// TwinCAT 3 PLC project PLC1
// ProgramVersion: 3.1.4024.0
// libraries:
//   Tc2_Standard, * (Beckhoff Automation GmbH)
//   Tc2_System, * (Beckhoff Automation GmbH)
//   Tc2_Utilities, * (Beckhoff Automation GmbH)
//   Tc3_IotBase, * (Beckhoff Automation GmbH)
//   Tc3_Module, * (Beckhoff Automation GmbH)
//   Util, * (System)
// project tree:
//   CSL/Enums/ E_Step.TcTLEO
//   CSL/FB/IO/ FB_UpdateInputs.TcPOU, FB_UpdateOutputs.TcPOU, FB_UpdatesParams.TcPOU
//   CSL/FB/Main/ FB_CSL_MAIN.TcPOU, FB_Oscillator.TcPOU, FB_Restore.TcPOU
//   CSL/FB/Piston/ FB_MSF_Pistons.TcPOU
//   CSL/FB/Sensor/ FB_Filter.TcPOU (not stored), FB_Measuring.TcPOU, FB_MSF_Sensor.TcPOU, FB_Processing.TcPOU
//   CSL/FC/ FC_Conversion.TcPOU, FC_thresholdsCalculation.TcPOU
//   CSL/Structs/ ST_CSL_RawOut.TcDUT (not stored), ST_CSL_In.TcDUT (not stored), ST_CSL_Out.TcDUT (not stored), ST_CSL_Params.TcDUT, ST_CSL_RawIn.TcDUT, ST_HMI_In.TcDUT, ST_HMI_Out.TcDUT, ST_HMI_Params.TcDUT
//   GVLs/ GVL_IOT.TcGVL, GVL_PLC.TcGVL
//   / IoTTask.TcTTO, PlcTask.TcTTO
//   IOT/Enums/ E_IOT_DataType.TcDUT, E_IOT_Step.TcDUT, E_IOT_UpdateSpeed.TcDUT
//   IOT/ FB_IOT.TcPOU, GVL_IOT_Constants.TcGVL
//   IOT/Functions/ F_IOT_GetPayload.TcPOU, F_IOT_IsValueEqual.TcPOU
//   IOT/Structs/ ST_IOT_Data.TcDUT, ST_IOT_OnChangePublishData.TcDUT, ST_IOT_Params.TcDUT, ST_IOT_PeriodicPublishData.TcDUT
//   IOT/Unions/ U_IOT_DataValue.TcDUT
//   POUs/ IOT_MAIN.TcPOU, MAIN.TcPOU
// real-time tasks:
//   TASK PlcTask: cycle T#10ms, priority 20, ADS port 350
//   TASK IoTTask: cycle T#10ms, priority 21, ADS port 351
// motion (NC):
//   TASK NC-Task 1 SAF: cycle T#2ms, priority 4, ADS port 501
//   TASK NC-Task 1 SVB: cycle T#10ms, priority 8, ADS port 511
//   AXIS Asse 1 (id 1)
//     OtherSettings: AllowMotionCmdToSlave=true
//     encoder EncType=4
//       EncPara: MaxCount=#x0000ffff
//         Inc: RefSoftSyncMask=#x0000ffff
//     drive DrvType=24
//       Analog: TorqueSetpointScale=10, ScaleFactorActTorque=0.1
//       TimeComp: TaskDelayCycles=1
//     controller CtrType=1
//       CtrPara: PriorControlFactor=1
//         Observer: BandWidth=20
//   AXIS Asse 2 (id 2)
//     OtherSettings: AllowMotionCmdToSlave=true
//     encoder EncType=4
//       EncPara: MaxCount=#x0000ffff
//         Inc: RefSoftSyncMask=#x0000ffff
//     drive DrvType=24
//       Analog: TorqueSetpointScale=10, ScaleFactorActTorque=0.1
//       TimeComp: TaskDelayCycles=1
//     controller CtrType=1
//       CtrPara: PriorControlFactor=1
//         Observer: BandWidth=20
//   AXIS Asse 3 (id 3)
//     OtherSettings: AllowMotionCmdToSlave=true
//     encoder EncType=4
//       EncPara: MaxCount=#x0000ffff
//         Inc: RefSoftSyncMask=#x0000ffff
//     drive DrvType=24
//       Analog: TorqueSetpointScale=10, ScaleFactorActTorque=0.1
//       TimeComp: TaskDelayCycles=1
//     controller CtrType=1
//       CtrPara: PriorControlFactor=1
//         Observer: BandWidth=20
// I/O:
//   DEVICE Dispositivo 1 (EtherCAT), AmsNetId 5.85.197.242.2.1
//     Terminale 1 (EK1200) [EK1200-5000 EtherCAT Power supply (2A E-Bus)]
//       Terminale 2 (EL1809) [EL1809 16Ch. Dig. Input 24V, 3ms]
//       Terminale 3 (EL2809) [EL2809 16Ch. Dig. Output 24V, 0.5A]
//       Terminale 4 (EL3201) [EL3201 1Ch. Ana. Input PT100 (RTD)]
//       Terminale 5 (EL3311) [EL3311 1Ch. Ana. Input Thermocouple (TC)]
//       Terminale 6 (EL3004) [EL3004 4Ch. Ana. Input +/-10V]
//       Terminale 7 (EL1918) [EL1918, 8Ch. Safety Input 24V, TwinSAFE]
//         modules: Module 1 (FSOE), Module 2 (FSLOGIC)
//       Terminale 8 (EL2904) [EL2904, 4 Ch. Safety Output 24V, 0.5A, TwinSAFE]
//         modules: Module 1 (FSOES), Module 2 (DO)
//       Terminale 9 (EL9011) [EL9011 End Terminal]
//   DEVICE Dispositivo 4 (EtherCAT), AmsNetId 5.85.197.242.5.1
//     Terminale 10 (EK1100) [EK1100 EtherCAT Coupler (2A E-Bus)]
//       Terminale 11 (EL1809) [EL1809 16Ch. Dig. Input 24V, 3ms]
//       Terminale 12 (EL2809) [EL2809 16Ch. Dig. Output 24V, 0.5A]
//       Terminale 13 (EL1809) [EL1809 16Ch. Dig. Input 24V, 3ms]
//       Terminale 14 (EL2809-0015) [EL2809-0015 16Ch. Dig. Output 24V DC, 0.35A, not short-circuit proof]
//       Terminale 15 (EL3202) [EL3202 2Ch. Ana. Input PT100 (RTD)]
//       Terminale 16 (EL3312) [EL3312 2Ch. Ana. Input Thermocouple (TC)]
//       Terminale 17 (EL3632) [EL3632 2Ch. IEPE Sensor]
//       Terminale 18 (EL7031) [EL7031 1Ch. Stepper motor output stage (24V, 1.5A)]
//       Terminale 10 (EL9011) [EL9011 End Terminal]
// variable links:
//   NC-Task 1 SAF/Axes/Asse 3 <-> Device 4 (EtherCAT)/Term 10 (EK1100)/Term 18 (EL7031)
//     Drive/Inputs/In/nState1 @bit 3 <-> STM Status/Status/Error
//     Drive/Inputs/In/nState1 @bit 5 <-> STM Status/Status/Moving negative
//     Drive/Inputs/In/nState1 @bit 4 <-> STM Status/Status/Moving positive
//     Drive/Inputs/In/nState1 @bit 1 <-> STM Status/Status/Ready
//     Drive/Inputs/In/nState1 <-> STM Status/Status/Ready to enable
//     Drive/Inputs/In/nState1 @bit 6 <-> STM Status/Status/Torque reduced
//     Drive/Inputs/In/nState1 @bit 2 <-> STM Status/Status/Warning
//     Drive/Inputs/In/nState2 @bit 3 <-> STM Status/Status/Digital input 1
//     Drive/Inputs/In/nState2 @bit 4 <-> STM Status/Status/Digital input 2
//     Drive/Inputs/In/nState2 @bit 5 <-> STM Status/Status/Sync error
//     Drive/Inputs/In/nState2 @bit 7 <-> STM Status/Status/TxPDO Toggle
//     Drive/Inputs/In/nState4 @bit 1 <-> WcState/InputToggle
//     Drive/Inputs/In/nState4 <-> WcState/WcState
//     Drive/Outputs/Out/nCtrl1 <-> STM Control/Control/Enable
//     Drive/Outputs/Out/nCtrl1 @bit 2 <-> STM Control/Control/Reduce torque
//     Drive/Outputs/Out/nCtrl1 @bit 1 <-> STM Control/Control/Reset
//     Drive/Outputs/Out/nDataOut2[0] <-> STM Velocity/Velocity
//     Enc/Inputs/In/nDataIn1[0] <-> ENC Status compact/Counter value
//     Enc/Inputs/In/nDataIn2[0] <-> ENC Status compact/Latch value
//     Enc/Inputs/In/nState1 @bit 4 <-> ENC Status compact/Status/Counter overflow
//     Enc/Inputs/In/nState1 @bit 3 <-> ENC Status compact/Status/Counter underflow
//     Enc/Inputs/In/nState1 @bit 1 <-> ENC Status compact/Status/Latch extern valid
//     Enc/Inputs/In/nState1 @bit 2 <-> ENC Status compact/Status/Set counter done
//     Enc/Inputs/In/nState2 @bit 4 <-> ENC Status compact/Status/Status of extern latch
//     Enc/Inputs/In/nState2 @bit 5 <-> ENC Status compact/Status/Sync error
//     Enc/Inputs/In/nState2 @bit 7 <-> ENC Status compact/Status/TxPDO Toggle
//     Enc/Inputs/In/nState4 @bit 1 <-> WcState/InputToggle
//     Enc/Inputs/In/nState4 <-> WcState/WcState
//     Enc/Outputs/Out/nCtrl1 @bit 3 <-> ENC Control compact/Control/Enable latch extern on negative edge
//     Enc/Outputs/Out/nCtrl1 @bit 1 <-> ENC Control compact/Control/Enable latch extern on positive edge
//     Enc/Outputs/Out/nCtrl1 @bit 2 <-> ENC Control compact/Control/Set counter
//     Enc/Outputs/Out/nDataOut1[0] <-> ENC Control compact/Set counter value
//   PLC1/PLC1 Instance <-> Device 1 (EtherCAT)/Term 1 (EK1200)/Term 2 (EL1809)
//     PlcTask Inputs/MAIN.stRawIn.bAck <-> Channel 10/Input
//     PlcTask Inputs/MAIN.stRawIn.bEmerg <-> Channel 11/Input
//     PlcTask Inputs/MAIN.stRawIn.bMotorImpulse <-> Channel 1/Input
//     PlcTask Inputs/MAIN.stRawIn.bPieceSensorInput <-> Channel 2/Input
//     PlcTask Inputs/MAIN.stRawIn.bPieceSensorOutput <-> Channel 3/Input
//     PlcTask Inputs/MAIN.stRawIn.bSlot1 <-> Channel 5/Input
//     PlcTask Inputs/MAIN.stRawIn.bSlot2 <-> Channel 6/Input
//     PlcTask Inputs/MAIN.stRawIn.bSlot3 <-> Channel 7/Input
//     PlcTask Inputs/MAIN.stRawIn.bStart <-> Channel 8/Input
//     PlcTask Inputs/MAIN.stRawIn.bStop <-> Channel 9/Input
//   PLC1/PLC1 Instance <-> Device 1 (EtherCAT)/Term 1 (EK1200)/Term 3 (EL2809)
//     PlcTask Outputs/MAIN.stRawOut.bCompressor <-> Channel 2/Output
//     PlcTask Outputs/MAIN.stRawOut.bLAck <-> Channel 8/Output
//     PlcTask Outputs/MAIN.stRawOut.bLStart <-> Channel 6/Output
//     PlcTask Outputs/MAIN.stRawOut.bLStop <-> Channel 7/Output
//     PlcTask Outputs/MAIN.stRawOut.bMotor <-> Channel 1/Output
//     PlcTask Outputs/MAIN.stRawOut.bValveSlot1 <-> Channel 3/Output
//     PlcTask Outputs/MAIN.stRawOut.bValveSlot2 <-> Channel 4/Output
//     PlcTask Outputs/MAIN.stRawOut.bValveSlot3 <-> Channel 5/Output
//   PLC1/PLC1 Instance <-> Device 1 (EtherCAT)/Term 1 (EK1200)/Term 6 (EL3004)
//     PlcTask Inputs/MAIN.stRawIn.nColorSensor <-> AI Standard Channel 1/Value

CONFIGURATION PLC1
    RESOURCE PLC ON TwinCAT3
        TASK IoTTask(INTERVAL := T#10ms, PRIORITY := 21);
        TASK PlcTask(INTERVAL := T#10ms, PRIORITY := 20);
        PROGRAM IOT_MAIN WITH IoTTask : IOT_MAIN;
        PROGRAM MAIN WITH PlcTask : MAIN;
    END_RESOURCE
END_CONFIGURATION

// ---- CSL/Enums/E_Step.TcTLEO
{attribute 'qualified_only'}
{attribute 'strict'}
{attribute 'to_string'}
TYPE E_Step :
(
	(* special steps *)
	NoStep := -32767,  // No step   
	Unknown := -32000, // unknown step
	
	(* Not Enabled or Errors*)    
	NeOrError := -990, // Not Enabled or Errors
	
	(*MSF Steps*)
	//main steps
	MainStop 		:= 	10, 		// stop
	MainSensor		:=	20,		// sensor area
	MainPiston		:=	30,		// piston area
	MainPause		:=	40,		// pause
	MainEmergency	:=	50,		// emergency
	MainAcknowledge	:=	60,		// acknowledge
	//sub-steps
	Stop			:=  90,
	Start			:= 	100,
	Measuring		:= 	110,
	Processing		:= 	120,
	conveyor		:=  130,	// a new piece was placed on the conveyor belt
	waiting			:= 	140,	// attesa
	piston			:=	150		// pistone

);
END_TYPE
//  NoStep = '-32767'
//  Unknown = '-32000'
//  NeOrError = '-990'

// ---- CSL/Structs/ST_CSL_Params.TcDUT
TYPE ST_CSL_Params :
STRUCT
	StepSlot1			:	INT		:= 	3;  // conveyor steps to reach Slot 1
	StepSlot2			:	INT		:= 	8;  // conveyor steps to reach Slot 2
	StepSlot3			:	INT		:= 	13; // conveyor steps to reach Slot 3
	StepNoSlot			:	INT		:=	20; // unknown colour -> discard piece
		
	pistonReentryDelay	:	TIME	:= T#500MS; // piston re-entry time
	stopLongPressTime	:	TIME	:= T#500MS;	// time required for the pause transition to be activated
	slotRemoveTime		:	TIME	:= T#500MS; // time required after piece removal from its slot
	
	(*Colors Voltage*)
	RedVoltage			:	REAL;	//	:=	5.5;
	BlueVoltage			:	REAL;	//	:=	7.1;
	WhiteVoltage		:	REAL;	//	:=	2.9;
	
	//threshold
	Threshold			:	REAL;	//	:=	0.5;
	
	//min values
	RedVoltageMin		:	REAL;
	BlueVoltageMin		:	REAL;
	WhiteVoltageMin		:	REAL;
	
	//max values
	RedVoltageMax		:	REAL;
	BlueVoltageMax		:	REAL;
	WhiteVoltageMax		:	REAL;
	
	(*Colors Slot*)
	WhiteSlot			:	INT;	//	:=	1;
	BlueSlot			:	INT;	//	:=	2;
	RedSlot				:	INT;	//	:=	3;

END_STRUCT
END_TYPE

// ---- CSL/Structs/ST_CSL_RawIn.TcDUT
TYPE ST_CSL_RawIn :
STRUCT
	(*Digital Inputs*)
	bMotorImpulse 		AT %I*	:	BOOL;	//I1  (NC)
	bPieceSensorInput 	AT %I*	:	BOOL;	//I2  (NC)
	bPieceSensorOutput 	AT %I*	:	BOOL;	//I3  (NO)
	bSlot1 				AT %I*	:	BOOL;	//I5  (NC)
	bSlot2 				AT %I*	:	BOOL;	//I6  (NC)
	bSlot3				AT %I*	:	BOOL;	//I7  (NC)
	
	bStart 				AT %I*	:	BOOL;	//I9  (NO)
	bStop				AT %I*	:	BOOL;	//I10 (NC)
	bAck 				AT %I*	:	BOOL;	//I11 (NO)
	bEmerg 				AT %I*	:	BOOL;	//I12 (NC)
	bMainEmerg			AT %I*	:	BOOL;	//I13 (NC)
	
	(*Analog Input*)
	nColorSensor		AT %I*	:	INT;	//I4
END_STRUCT
END_TYPE

// ---- CSL/Structs/ST_HMI_In.TcDUT
TYPE ST_HMI_In :
STRUCT
	bStart 		:	BOOL;
	bStop 		:	BOOL;
	bAck		:	BOOL;
END_STRUCT
END_TYPE

// ---- CSL/Structs/ST_HMI_Out.TcDUT
TYPE ST_HMI_Out :
STRUCT
	bGreen	:BOOL;
	bRed	:BOOL;
	bOrange	:BOOL;
END_STRUCT
END_TYPE

// ---- CSL/Structs/ST_HMI_Params.TcDUT
TYPE ST_HMI_Params :
STRUCT
	(*Params*)
	//slot
	WhiteSlot		:	INT	:= 1;
	BlueSlot		:	INT	:= 2;
	RedSlot			:	INT := 3;
	
	//voltage levels
	RedVoltage		:	REAL	:= 5.5;
	BlueVoltage		:	REAL	:= 7.1;
	WhiteVoltage	:	REAL	:= 2.9;
	
	//threshold
	Threshold		:	REAL	:=	0.5;
END_STRUCT
END_TYPE

// ---- IOT/Enums/E_IOT_DataType.TcDUT
(* -----------------------------------------------------------------------------
| This sample has been supplied by Beckhoff As-Is and is intended only as an   |
| example implementation. Functionality is not guaranteed.                     |
----------------------------------------------------------------------------- *)

// questa enumerazione descrive serve per identificare il tipo di dato contenuto
// all'interno dell'unione U_IOT_DataValue in modo da poterlo interpretare 
// correttamente

{attribute 'qualified_only'}
{attribute 'strict'}
TYPE E_IOT_DataType :
(
	Boolean := 0,
	I32 := 1,
	F64 := 2,
	S50 := 51
);
END_TYPE

// ---- IOT/Enums/E_IOT_Step.TcDUT
(* -----------------------------------------------------------------------------
| This sample has been supplied by Beckhoff As-Is and is intended only as an   |
| example implementation. Functionality is not guaranteed.                     |
----------------------------------------------------------------------------- *)

// passi della macchina a stati che gestisce la comunicazione IOT

{attribute 'qualified_only'}
{attribute 'strict'}
TYPE E_IOT_Step :
(
	(* special steps *)
	NoStep := -32767,		// nessuno step
	Unknown := -32000,		// step sconosciuto
	
	(* Error steps *)
	NeOrError := -990,		// non abilitata o in errore
	Reset := -980,			// azzeramento errori

	(* Stop *)
	Stop := 0,				// stop
	
	(* Cycle *)
	Configure := 100,		// configurazione 
	Connect := 200,			// connessione
	Subscribe := 210,		// sottoscrivi i topic che interessano
	Online := 220,			// in linea
	Unsubscribe := 300,		// rimuovi sottoscrizioni
	Disconnect := 310		// disconnessione
);
END_TYPE

// ---- IOT/Enums/E_IOT_UpdateSpeed.TcDUT
(* -----------------------------------------------------------------------------
| This sample has been supplied by Beckhoff As-Is and is intended only as an   |
| example implementation. Functionality is not guaranteed.                     |
----------------------------------------------------------------------------- *)

// questa enumerazione serve ad identificare il periodo di aggiornamento dei
// dati che vengono pubblicati su MQTT

{attribute 'qualified_only'}
{attribute 'strict'}
TYPE E_IOT_UpdateSpeed :
(
	Slow := 0,			// 1s	
	Fast := 1			// 100ms
);
END_TYPE

// ---- IOT/Structs/ST_IOT_Data.TcDUT
(* -----------------------------------------------------------------------------
| This sample has been supplied by Beckhoff As-Is and is intended only as an   |
| example implementation. Functionality is not guaranteed.                     |
----------------------------------------------------------------------------- *)

// Questa struttura definisce il dato da pubblicare sul broker
// Ad ogni dato viene associato un subtopic specifico

TYPE ST_IOT_Data :
STRUCT
	sSubtopic : STRING;				// subtopic dove il valore verra scritto
	eType : E_IOT_DataType;			// tipologia del dato (DINT, LREAL, BOOL)
	uValue : U_IOT_DataValue;		// unione in cui viene letto/scritto il valore	
END_STRUCT
END_TYPE

// ---- IOT/Structs/ST_IOT_OnChangePublishData.TcDUT
(* -----------------------------------------------------------------------------
| This sample has been supplied by Beckhoff As-Is and is intended only as an   |
| example implementation. Functionality is not guaranteed.                     |
----------------------------------------------------------------------------- *)

// Questa struttura definisce un dato da pubblicare al cambiamento del suo
// valore. Oltre al dato è presente nellea struttura l'elemento che su cui
// salvare il valore precedente in modo da poter fare dei confronti

TYPE ST_IOT_OnChangePublishData :
STRUCT
	uOldValue : U_IOT_DataValue;
	stData : ST_IOT_Data;		
END_STRUCT
END_TYPE

// ---- IOT/Structs/ST_IOT_Params.TcDUT
(* -----------------------------------------------------------------------------
| This sample has been supplied by Beckhoff As-Is and is intended only as an   |
| example implementation. Functionality is not guaranteed.                     |
----------------------------------------------------------------------------- *)

// Questa struttura cointiene i parametri necessari al funzionamento della
// FB_IOT. 

TYPE ST_IOT_Params :
STRUCT
	// i parametri per instaurare la connessione con il broker 
	//sHostName : STRING := 'test.mosquitto.org';
	sMQTTHostName : STRING := 'item2122a.cloud.shiftr.io';
	nHostPort : UINT := 1883; 
	// Si possono usare anche user e password. 
    // vd: https://infosys.beckhoff.com/content/1033/tf6701_tc3_iot_communication_mqtt/3391835403.html?id=6531035858226877065
	sUserName : STRING := 'item2122a';
	sUserPassword : STRING := 'K2Xpe5XV3yvL7zcu';
	
	// certificati necessari per l'autenticazione. 
	stMqttTls : ST_IotMqttTls := ();
		
	// topic generale all'interno del quale ci saranno i subtopic nei quali
	// verranno pubblicati i dati
	// il pragma {attribute 'TcEncoding':='UTF-8'} va sempre usato per le 
	// stringhe quando si opera con MQTT
	{attribute 'TcEncoding':='UTF-8'}
	sTopicPrefix : STRING := 'ColorSorter';
	
	// subtopic da sottoscrivere per leggere i comandi  
	{attribute 'TcEncoding':='UTF-8'}
	sCmdSubscribedTopic : STRING := '/cmd';
	
	// numero massimo di messaggi da leggere per ciclo dai topic sottoscritti 
	nDequeueMessagesPerCycle : UINT := 3;
END_STRUCT
END_TYPE

// ---- IOT/Structs/ST_IOT_PeriodicPublishData.TcDUT
(* -----------------------------------------------------------------------------
| This sample has been supplied by Beckhoff As-Is and is intended only as an   |
| example implementation. Functionality is not guaranteed.                     |
----------------------------------------------------------------------------- *)

// Questa struttura definisce un dato da pubblicare ciclicamente. Oltre al 
// dato è presente nellea struttura l'elemento che definisce l'intervallo 
// di pubblicazione

TYPE ST_IOT_PeriodicPublishData :
STRUCT
	eUpdateSpeed : E_IOT_UpdateSpeed;
	stData : ST_IOT_Data;	
END_STRUCT
END_TYPE

// ---- IOT/Unions/U_IOT_DataValue.TcDUT
(* -----------------------------------------------------------------------------
| This sample has been supplied by Beckhoff As-Is and is intended only as an   |
| example implementation. Functionality is not guaranteed.                     |
----------------------------------------------------------------------------- *)

// Questa unione contiene il valore del dato. L'utilizzo dell'unione permette
// di avere una struttura dato (ST_IOT_Data) generica evitando di preoccuparsi 
// di quale sia il tipo di dato contenuto se non quando si va effettivamente 
// a leggerlo o scriverlo.
// La quantità di memoria occupata da una union corrisponde alla quantita di 
// memoria necessaria a contenere l'elemento della union che da dimensione
// maggiore.
// In sostanza i vari elementi di una union condividono la stessa area di
// memoria e usarne uno piuttosto di un altro non modifica il contenuto della
// memoria stessa quanto la sua rappresentazione.

TYPE U_IOT_DataValue :
UNION
	b : BOOL;
	n : DINT;
	f : LREAL;
	sv : STRING(50);
END_UNION
END_TYPE

// ---- GVLs/GVL_IOT.TcGVL
(* -----------------------------------------------------------------------------
| This sample has been supplied by Beckhoff As-Is and is intended only as an   |
| example implementation. Functionality is not guaranteed.                     |
----------------------------------------------------------------------------- *)

{attribute 'qualified_only'}
VAR_GLOBAL PERSISTENT
	stIotParams : ST_IOT_Params;		// Parametri per la comunicazione MQTT
//	stFlmCmd : ST_FLM_Cmd;				// comandi di FLM
END_VAR

// ---- GVLs/GVL_PLC.TcGVL
{attribute 'qualified_only'}
VAR_GLOBAL
	strEStep	:	STRING;
	strEsubStepSensor	:	STRING;
	strEsubStepPiston	:	STRING;
	
	estep 	: E_Step;
	eSubStepSensor: E_Step;
	eSubStepPistons: E_Step;
	
	nColorSensor	:	REAL;
	
	nTotalRevs		:	REAL;
	
	nCycles			:	INT;
END_VAR

// ---- IOT/GVL_IOT_Constants.TcGVL
(* -----------------------------------------------------------------------------
| This sample has been supplied by Beckhoff As-Is and is intended only as an   |
| example implementation. Functionality is not guaranteed.                     |
----------------------------------------------------------------------------- *)


{attribute 'qualified_only'}
VAR_GLOBAL CONSTANT
	cIOTMAXDATA : UDINT := 32;
END_VAR

// ---- POUs/IOT_MAIN.TcPOU
(* -----------------------------------------------------------------------------
| This sample has been supplied by Beckhoff As-Is and is intended only as an   |
| example implementation. Functionality is not guaranteed.                     |
----------------------------------------------------------------------------- *)

PROGRAM IOT_MAIN
VAR
	bInitialized : BOOL;
	bConnect : BOOL;		// richiesta TRUE -> connetti FALSE -> disconnetti
	
	// array per i dati da pubblicare e loro dimensione 
	aPeriodicPublish : ARRAY[0..GVL_IOT_Constants.cIOTMAXDATA - 1] OF ST_IOT_PeriodicPublishData;
	aOnChangePublish : ARRAY[0..GVL_IOT_Constants.cIOTMAXDATA - 1] OF ST_IOT_OnChangePublishData;		
	nPeriodicPublishSize : UDINT;	
	nOnChangePublishSize : UDINT;	
	
	fbIot : FB_IOT;
	nInitCycles : UDINT;
END_VAR

(* -----------------------------------------------------------------------------
| This sample has been supplied by Beckhoff As-Is and is intended only as an   |
| example implementation. Functionality is not guaranteed.                     |
----------------------------------------------------------------------------- *)

IF NOT bInitialized THEN
	IF nInitCycles = 0 THEN	
		ACT_InitPeriodic();	
		ACT_InitOnChange();
	END_IF;
	nInitCycles := nInitCycles + 1;
	bConnect := TRUE;
	bInitialized := (GVL_PLC.estep = E_Step.MainStop );
ELSE
	
	// Qui vengono letti ad ogni ciclo i valori da FLM che verranno pubblicati
	// nei topic corrispondenti
 
//	aOnChangePublish[0].stData.uValue.n := TO_DINT(GVL_PLC.stFlmStatus.eStep);
//	aOnChangePublish[1].stData.uValue.b := GVL_PLC.stFlmStatus.bFailure;
//	aOnChangePublish[2].stData.uValue.b := GVL_PLC.stFlmStatus.bWarning;

    aOnChangePublish[0].stData.uValue.f := TO_REAL(GVL_PLC.nColorSensor);
    aOnChangePublish[1].stData.uValue.sv := GVL_PLC.strEStep;
    aOnChangePublish[2].stData.uValue.sv := GVL_PLC.strEsubStepSensor;	
    aOnChangePublish[3].stData.uValue.sv := GVL_PLC.strEsubStepPiston;	
	aOnChangePublish[4].stData.uValue.f := GVL_PLC.nTotalRevs;	
	aOnChangePublish[5].stData.uValue.n := GVL_PLC.nCycles;
	
//	aPeriodicPublish[0].stData.uValue.b := GVL_PLC.stFlmOut.bCorkingVertical;

	
	fbIot(
		bEnable:= TRUE, 
		bConnect:= bConnect, 
		tAutoAckTime:= T#2M, 
		stParams:= GVL_IOT.stIotParams, 
		aPeriodicPublish := aPeriodicPublish,		
		aOnChangePublish := aOnChangePublish,
		nPeriodicPublishSize := nPeriodicPublishSize, 
		nOnChangePublishSize := nOnChangePublishSize
	);
	
	// I comandi letti nel subtopic corrispondente vengono qui scritti su
	// delle variabili globali in modo da poter essere letti dalla task PLC
	// e usati all'interno di FLM
//	GVL_IOT.stFlmCmd.bStart := fbIot.bFlmStartCmd;
//	GVL_IOT.stFlmCmd.bStop := fbIot.bFlmStopCmd;
//	GVL_IOT.stFlmCmd.bAck := fbIot.bFlmAckCmd;
END_IF

ACTION ACT_InitOnChange:
(* -----------------------------------------------------------------------------
| This sample has been supplied by Beckhoff As-Is and is intended only as an   |
| example implementation. Functionality is not guaranteed.                     |
----------------------------------------------------------------------------- *)

// inizializzazione degli elementi dell'array che contiene i dati da scambiare
// al cambiamento

aOnChangePublish[0].stData.sSubtopic := '/ncolorsensor';
aOnChangePublish[0].stData.eType := E_IOT_DataType.F64;

aOnChangePublish[1].stData.sSubtopic := '/estep';
aOnChangePublish[1].stData.eType := E_IOT_DataType.S50;

aOnChangePublish[2].stData.sSubtopic := '/esubstepsensor';
aOnChangePublish[2].stData.eType := E_IOT_DataType.S50;

aOnChangePublish[3].stData.sSubtopic := '/esubsteppistons';
aOnChangePublish[3].stData.eType := E_IOT_DataType.S50;

aOnChangePublish[4].stData.sSubtopic := '/nTotalRevs';
aOnChangePublish[4].stData.eType := E_IOT_DataType.F64;

aOnChangePublish[5].stData.sSubtopic := '/nCycles';
aOnChangePublish[5].stData.eType := E_IOT_DataType.I32;

//aOnChangePublish[2].stData.sSubtopic := '/Warning';
//aOnChangePublish[2].stData.eType := E_IOT_DataType.Boolean;

// dimensione effettiva dell'array
nOnChangePublishSize := 6;
END_ACTION

ACTION ACT_InitPeriodic:
(* -----------------------------------------------------------------------------
| This sample has been supplied by Beckhoff As-Is and is intended only as an   |
| example implementation. Functionality is not guaranteed.                     |
----------------------------------------------------------------------------- *)

// inizializzazione degli elementi dell'array che contiene i dati da scambiare
// ciclicamente.

aPeriodicPublish[0].eUpdateSpeed := E_IOT_UpdateSpeed.Fast;
aPeriodicPublish[0].stData.sSubtopic := '/TaskRunning';
aPeriodicPublish[0].stData.eType := E_IOT_DataType.Boolean;

(*
aPeriodicPublish[1].eUpdateSpeed := E_IOT_UpdateSpeed.Fast;
aPeriodicPublish[1].stData.sSubtopic := '/CorkingRotation';
aPeriodicPublish[1].stData.eType := E_IOT_DataType.Boolean;

aPeriodicPublish[2].eUpdateSpeed := E_IOT_UpdateSpeed.Slow;
aPeriodicPublish[2].stData.sSubtopic := '/WaterLevel';
aPeriodicPublish[2].stData.eType := E_IOT_DataType.F64;

aPeriodicPublish[3].eUpdateSpeed := E_IOT_UpdateSpeed.Slow;
aPeriodicPublish[3].stData.sSubtopic := '/MintLevel';
aPeriodicPublish[3].stData.eType := E_IOT_DataType.F64;
*)

// dimensione effettiva dell'array
nPeriodicPublishSize := 1;
END_ACTION

END_PROGRAM

// ---- IOT/FB_IOT.TcPOU
(* -----------------------------------------------------------------------------
| This sample has been supplied by Beckhoff As-Is and is intended only as an   |
| example implementation. Functionality is not guaranteed.                     |
----------------------------------------------------------------------------- *)

FUNCTION_BLOCK FB_IOT

VAR_INPUT
	bEnable : BOOL;						// abilitazione della FB
	bConnect : BOOL;					// bit che richiede la connessione
	tAutoAckTime : TIME;				// tempo di auto riconoscimento degli errori
	stParams : ST_IOT_Params;			// parametri 
	nPeriodicPublishSize : UDINT;		// dimensione dell'array che continene i dati da pubblicare a tempo
	nOnChangePublishSize : UDINT;		// dimensione dell'arra che contiene i dati da pubblicare al cambiamento
END_VAR

VAR_IN_OUT
	aPeriodicPublish : ARRAY[0..GVL_IOT_Constants.cIOTMAXDATA - 1] OF ST_IOT_PeriodicPublishData;	// array di dati da pubblicare a tempo
	aOnChangePublish : ARRAY[0..GVL_IOT_Constants.cIOTMAXDATA - 1] OF ST_IOT_OnChangePublishData;	// array di dati da pubblicare al cambiamento
END_VAR

VAR_OUTPUT
	eStep :  E_IOT_Step;		// passo della macchina a stati
	tStepTime : TIME;			// tempo nel passo
	eErrStep : E_IOT_Step;		// passo in cui si è generato l'errore
	nErrId : DINT;				// id dell'errore
	bFlmStartCmd : BOOL;		// comando di start per FLM
	bFlmStopCmd : BOOL;			// comando di stop per FLM
	bFlmAckCmd : BOOL;			// comando di Ack per FLM
END_VAR

VAR
	bInitialized :  BOOL;
	eNewstep :  E_IOT_Step;
	bEntryact :  BOOL;
	fbTonStep :  TON;	
	bForceOnChangePublish : BOOL;	// forza la pubblicazione dei dati al cambiamento (acnhe se non sono cambiati)
	bMqttConnect : BOOL;			// bit di connessione MQTT
	udi : UDINT;
	fbMqttClient : FB_IotMqttClient;			// client MQTT	
	fbMessageQueue : FB_IotMqttMessageQueue;	// coda dei messaggi in ingresso	
	fbMessage : FB_IotMqttMessage;				// messaggio
	sPayload : STRING(255);
	bIsEqual : BOOL;	
	fbBlinkFast : BLINK;						// blink per la pubblicazione dati veloci
	fbBlinkSlow : BLINK;						// blinck pubblicazione dati lenti
	fbRtFast : R_TRIG;							// trigger pubblicazione dati veloci
	fbRtSlow : R_TRIG;							// trigger pubblicazione dati lenti
	bCmdTopicSubscribed : BOOL;	
	nDequeueCnt : UINT := 0;					// contatore di scodamento
	{attribute 'TcEncoding':='UTF-8'}
	sTopicRcv : STRING(255);					
	{attribute 'TcEncoding':='UTF-8'}
	sPayloadRcv : STRING(255);	
	{attribute 'TcEncoding':='UTF-8'}
	sAppo: STRING(255);	
	nFlmCmd : UINT := 0;
	fbTpFlmStartCmd : TP;						// impulso comando start FLM
	fbTpFlmStopCmd : TP;						// impulso comando start FLM
	fbTpFlmAckCmd : TP;							// impulso comando start FLM
END_VAR

(* -----------------------------------------------------------------------------
| This sample has been supplied by Beckhoff As-Is and is intended only as an   |
| example implementation. Functionality is not guaranteed.                     |
----------------------------------------------------------------------------- *)

// Questa macchina a stati serve per gestire la connessione verso il broker,
// la pubblicazione dei dati e la lettura dei messaggi nei topic sottoscritti.
// Tutto si basa su una FB di tipo FB_IotMqttClient
// https://infosys.beckhoff.com/content/1033/tf6701_tc3_iot_communication_mqtt/3391835403.html?id=6531035858226877065
// FB_IotMqttClient utilizza il paradigma della programmazione ad oggetti
// e in sostanza è una classe. Senza addentrarsi in una spiegazione della
// programmazione ad oggetti basti dire che una istanza di questa FB è un
// oggetto sul quale possono essere chiamati dei metodi. I metodi sono delle 
// funzioni proprie dell'oggetto specifico (l'istanza di FB_IotMqttClient) che
// hanno visibilità sulle variabili locali dell'oggetto. Ciascun metodo ha 
// la sua uscita, i suoi ingressi e le sue proprie variabili locali (temporanee)
// ma può anche operare sulle variabili locali dell'oggetto (l'istanza) che non 
// sono temporanee ma mantengono il valore tra una chiamata e l'altra. In 
// questo modo metodi diversi possono condividere delle aree di memoria che 
// altro non è che quella definita nelle variabili locali dell'oggetto.


IF NOT bInitialized THEN
	eNewstep := E_IOT_Step.NoStep;
	eStep := E_IOT_Step.Stop;
	bEntryact := FALSE;
	bInitialized := TRUE;		
ELSE	
	(* disabilitata o avaria *)	
	IF NOT bEnable THEN
		eNewstep := E_IOT_Step.NeOrError;
	END_IF
	
	IF eNewstep <> E_IOT_Step.NoStep THEN
		eStep := eNewstep;
		eNewstep := E_IOT_Step.NoStep;
		bEntryact := FALSE;
	END_IF;

	(* filtri *)	
	
	(* fronti *)	
	
	// questi blink e trigger servono a creare due bit (i trigger fast e slow)
	// che sono a TRUE solo per un ciclo ogni, rispettivamente, 100ms e 1s
	fbBlinkFast(ENABLE:= TRUE, TIMELOW:= T#50MS , TIMEHIGH:= T#50MS);	
	fbBlinkSlow(ENABLE:= TRUE, TIMELOW:= T#5S , TIMEHIGH:= T#5S);
	fbRtFast(CLK := fbBlinkFast.OUT);	
	fbRtSlow(CLK := fbBlinkSlow.OUT);
	
	(* richieste *)
	
	CASE eStep OF
		
		(* not Enabled or Error *)
		E_IOT_Step.NeOrError :
			(* entry action *)
			IF NOT bEntryact THEN
				bEntryact := TRUE;
			END_IF;

			(* body *)
			bMqttConnect := FALSE;
			bCmdTopicSubscribed := FALSE;
					
			(* transition *)
			IF bEnable THEN	
				IF tStepTime > tAutoAckTime THEN 		
					// qui si fa sostanzialmente un autoreset invece che lasciare 
					// tutto bloccato fino ad un intervento umano. Questa scelta si 
					// può fare per le funzionalitàù di comunicazione ma va sempre 
					// ben ponderata. Qui per esempio si valuta che è preferibile 
					// tentare di riconnettersi e che perdere informazioni sulle 
					// casuse di errore non è molto importante.
					eNewstep := E_IOT_Step.Reset;
				END_IF
			END_IF

			(* exitact *)
			IF eNewstep <> E_IOT_Step.NoStep THEN
				nErrId := 0;
				eErrStep := E_IOT_Step.NoStep;
			END_IF;

		(* Reset *)
		E_IOT_Step.Reset :
			(* entry action *)
			IF NOT bEntryact THEN				
				bEntryact := TRUE;
			END_IF;

			(* body *)
			bMqttConnect := FALSE;
					
			(* transition *)
			IF bEnable THEN				
				eNewstep := E_IOT_Step.Stop;				
			END_IF

			(* exitact *)
			IF eNewstep <> E_IOT_Step.NoStep THEN
				;
			END_IF;		
			
		(* Stop *)
		E_IOT_Step.Stop:
			(* entry action *)
			IF NOT bEntryact THEN
				bEntryact := TRUE;
			END_IF;

			(* body *)
			bMqttConnect := FALSE;			
							
			(* transition *)
			IF fbMqttClient.bError THEN
				eNewstep := E_IOT_Step.NeOrError;
			ELSE			
				IF bConnect THEN
					eNewstep := E_IOT_Step.Configure;
				END_IF
			END_IF
			
			(* exitact *)
			IF eNewstep <> E_IOT_Step.NoStep THEN
				IF eNewstep = E_IOT_Step.NeOrError THEN
					eErrStep := eStep;
					nErrID := fbMqttClient.hrErrorCode;				
				END_IF
			END_IF;
			
		(* Configure *)
		E_IOT_Step.Configure:
			(* entry action *)
			IF NOT bEntryact THEN
				bEntryact := TRUE;
			END_IF;

			(* body *)			
			fbMqttClient.sHostName:= stParams.sMQTTHostName;
			fbMqttClient.nHostPort:= stParams.nHostPort;
			fbMqttClient.sUserName:= stParams.sUserName;
			fbMqttClient.sUserPassword:= stParams.sUserPassword;
			//fbMqttClient.sClientId:= 'FLM'; 
			fbMqttClient.sTopicPrefix:= stParams.sTopicPrefix; 			 
			fbMqttClient.stTLS:= stParams.stMqttTls;
			fbMqttClient.nKeepAlive := 30;			
			fbMqttClient.ipMessageQueue := fbMessageQueue;			// FB che gestisce la coda di messaggi			
			bMqttConnect := FALSE;
							
			(* transition *)
			IF fbMqttClient.bError THEN
				eNewstep := E_IOT_Step.NeOrError;
			ELSE			
				eNewstep := E_IOT_Step.Connect;
			END_IF
			
			(* exitact *)
			IF eNewstep <> E_IOT_Step.NoStep THEN
				IF eNewstep = E_IOT_Step.NeOrError THEN
					eErrStep := eStep;
					nErrID := fbMqttClient.hrErrorCode;
				END_IF
			END_IF;
			
		(* Connect *)
		E_IOT_Step.Connect:
			(* entry action *)
			IF NOT bEntryact THEN
				bEntryact := TRUE;
			END_IF;

			(* body *)
			bMqttConnect := TRUE;
		
			(* transition *)
			IF fbMqttClient.bError THEN
				eNewstep := E_IOT_Step.NeOrError;
			ELSE
				IF bConnect THEN
					IF fbMqttClient.bConnected THEN
						eNewstep := E_IOT_Step.Subscribe;
					END_IF
				ELSE
					eNewstep := E_IOT_Step.Disconnect;	
				END_IF
			END_IF;
			
			(* exitact *)
			IF eNewstep <> E_IOT_Step.NoStep THEN
				IF eNewstep = E_IOT_Step.NeOrError THEN
					eErrStep := eStep;
					nErrID := fbMqttClient.hrErrorCode;
				END_IF
			END_IF;
			
		(* Subscribe *)
		E_IOT_Step.Subscribe:
			(* entry action *)
			IF NOT bEntryact THEN
				bCmdTopicSubscribed := FALSE;
				bEntryact := TRUE;
			END_IF;

			(* body *)
			bMqttConnect := TRUE;
			
			// questo metodo realizza la sottoscrizione al topic indicato
			// con la qualità del servizio indicata. 
			// (per QoS vedi: https://mosquitto.org/man/mqtt-7.html)
			bCmdTopicSubscribed := fbMqttClient.Subscribe(
				sTopic:=stParams.sCmdSubscribedTopic, 
				eQoS:=TcIotMqttQos.AtMostOnceDelivery			// qualità del servizo
			);
		
			(* transition *)
			IF fbMqttClient.bError OR NOT bCmdTopicSubscribed THEN
				eNewstep := E_IOT_Step.NeOrError;
			ELSE
				IF fbMqttClient.bConnected THEN
					eNewstep := E_IOT_Step.Online;
				END_IF
			END_IF;
			
			(* exitact *)
			IF eNewstep <> E_IOT_Step.NoStep THEN
				IF eNewstep = E_IOT_Step.NeOrError THEN
					eErrStep := eStep;
					nErrID := fbMqttClient.hrErrorCode;
				END_IF
			END_IF;
			
		(* Online *)
		E_IOT_Step.Online:
			(* entry action *)
			IF NOT bEntryact THEN	
				bForceOnChangePublish := TRUE;		
				bEntryact := TRUE;
			END_IF;

			(* body *)
			bMqttConnect := TRUE;
			ACT_PublishPeriodic();		// pubblicazione dati periodici
			ACT_PublishOnChange();		// pubblicazione dati al cambiamento
			ACT_DequeueMessages();		// lettura dei messaggi nei topic sottoscritti
		
			(* transition *)
			IF fbMqttClient.bError THEN
				eNewstep := E_IOT_Step.NeOrError;
			ELSE
				IF NOT bConnect THEN
					eNewstep := E_IOT_Step.Disconnect;
				END_IF
			END_IF;
			
			(* exitact *)
			IF eNewstep <> E_IOT_Step.NoStep THEN				
				IF eNewstep = E_IOT_Step.NeOrError THEN
					eErrStep := eStep;
					nErrID := fbMqttClient.hrErrorCode;
				END_IF
			END_IF;
			
		(* Unsubscribe *)
		E_IOT_Step.Unsubscribe:
			(* entry action *)
			IF NOT bEntryact THEN
				bCmdTopicSubscribed := FALSE;
				bEntryact := TRUE;
			END_IF;

			(* body *)
			bMqttConnect := TRUE;
			bCmdTopicSubscribed := NOT fbMqttClient.Unsubscribe(
				sTopic:=stParams.sCmdSubscribedTopic,				
			);
		
			(* transition *)
			IF fbMqttClient.bError OR NOT bCmdTopicSubscribed THEN
				eNewstep := E_IOT_Step.NeOrError;
			ELSE
				IF NOT bCmdTopicSubscribed THEN
					eNewstep := E_IOT_Step.Disconnect;
				END_IF
			END_IF;
			
			(* exitact *)
			IF eNewstep <> E_IOT_Step.NoStep THEN
				IF eNewstep = E_IOT_Step.NeOrError THEN
					eErrStep := eStep;
					nErrID := fbMqttClient.hrErrorCode;
				END_IF
			END_IF;
			
		(* Disconnect *)
		E_IOT_Step.Disconnect:
			(* entry action *)
			IF NOT bEntryact THEN
				bEntryact := TRUE;
			END_IF;

			(* body *)
			bMqttConnect := FALSE;
		
			(* transition *)
			IF fbMqttClient.bError THEN
				eNewstep := E_IOT_Step.NeOrError;
			ELSE
				IF NOT fbMqttClient.bConnected THEN
					eNewstep := E_IOT_Step.Stop;
				END_IF
			END_IF;
			
			(* exitact *)
			IF eNewstep <> E_IOT_Step.NoStep THEN
				IF eNewstep = E_IOT_Step.NeOrError THEN
					eErrStep := eStep;
					nErrID := fbMqttClient.hrErrorCode;
				END_IF
			END_IF;			
		ELSE
			eNewstep := E_IOT_Step.NeOrError;
			eErrStep := E_IOT_Step.Unknown;
			nErrId := -9;			
	END_CASE;
	
	(* tempo di permanenza nello step *)
	fbTonStep(IN := (eNewstep = E_IOT_Step.NoStep), PT := T#500H);
	tStepTime := fbTonStep.ET;
	
	(* FBs *)
	// questo metodo Execute va richiamato ad ogni ciclo. Si occupa di
	// instaurare e mantenere la connessione fino a quando l'ingresso 
	// passato è a TRUE	
	fbMqttClient.Execute(bMqttConnect);
	
	(* uscite *)
	fbTpFlmStartCmd(IN:= nFlmCmd = 1, PT:= T#200MS);
	fbTpFlmStopCmd(IN:= nFlmCmd = 2, PT:= T#200MS);
	fbTpFlmAckCmd(IN:= nFlmCmd = 3, PT:= T#200MS);
	bFlmStartCmd := fbTpFlmStartCmd.Q;
	bFlmStopCmd := fbTpFlmStopCmd.Q;
	bFlmAckCmd := fbTpFlmAckCmd.Q;

	
END_IF;

ACTION ACT_DequeueMessages:
(* -----------------------------------------------------------------------------
| This sample has been supplied by Beckhoff As-Is and is intended only as an   |
| example implementation. Functionality is not guaranteed.                     |
----------------------------------------------------------------------------- *)

// Questa action si occupa di verificare se ci sono messaggi nei subtopic 
// sottoscritti ed eventualmente di leggerli e decodificarli. 
// fbMessageQueue era stata precedentemente passata ad fbMqttClient in questo
// modo la coda può essere gestita dall'interno di fbMqttClient e anche 
// all'esterno.
// A sua volta fbMessage, che è una FB che serve a gestire il singolo messaggio
// viene passata a fbMessageQueue in modo che il messaggio sia gestibile sia 
// dall'interno di fbMessageQueue che dall'esterno.
// Se presente il messaggio viene scodato con fbMessageQueue.Dequeue poi
// si vanno a leggere il Topic e il payload con fbMessage.GetTopic  e
// fbMessage.GetPayload. Successivamente si estrapola dal topic completo
// solo la parte di subtopic che ci interessa per verifcare che corrisponda 
// al subtopic che abbiamo impostato nei parametri e solo a questo punto, 
// in base al valore del payload si prendono le azioni corrispondenti impostando
// la variabile nFlm a tre valori codificati (NB qui sarebbe stata una 
// buona idea usare una enumerazione... pazienza)

nFlmCmd := 0;
FOR nDequeueCnt := 0 TO stParams.nDequeueMessagesPerCycle - 1 DO
	IF fbMessageQueue.nQueuedMessages > 0 THEN
		IF fbMessageQueue.Dequeue(fbMessage:=fbMessage) THEN
			fbMessage.GetTopic(
					pTopic:=ADR(sTopicRcv), 
					nTopicSize:=SIZEOF(sTopicRcv)
			);
			fbMessage.GetPayload(
				pPayload:=ADR(sPayloadRcv), 
				nPayloadSize:=SIZEOF(sPayloadRcv),
				bSetNullTermination:=TRUE
			);
			
			 FindAndDelete(
				pSrcString:= ADR(sTopicRcv), 
				pDeleteString:= ADR(stParams.sTopicPrefix), 
				pDstString:= ADR(sAppo), 
				nDstSize:= SIZEOF(sAppo)
			);
			
			IF sAppo = stParams.sCmdSubscribedTopic THEN
				IF sPayloadRcv = 'start' THEN
					nFlmCmd := 1;
				ELSIF sPayloadRcv = 'stop' THEN
					nFlmCmd := 2;
				ELSIF sPayloadRcv = 'ack' THEN
					nFlmCmd := 3;
				END_IF
			END_IF
		END_IF
	END_IF	
END_FOR
END_ACTION

ACTION ACT_PublishOnChange:
(* -----------------------------------------------------------------------------
| This sample has been supplied by Beckhoff As-Is and is intended only as an   |
| example implementation. Functionality is not guaranteed.                     |
----------------------------------------------------------------------------- *)

// Questa Action si occupa della pubblicazione dei dati al cambiamento. Si cicla 
// tra gli elementi dell'array verificando che il dato sia cambiato per mezzo 
// di F_IOT_IsValueEqual. Se il dato è cambiato oppure la pubblicazione è 
// forzata tramite bForceOnChangePublish viene calcolato il payload con 
// F_IOT_GetPayload che converte il valore del dato in una stringa
// e lo si pubblica sul topic con il metodo Public di fbMqttClient.
// L'ingresso eQos indica la qualità richiesta per questa pubblicazione: in
// questo caso si desidera che la pubblicazione avvenga una e una sola volta, 
// senza duplicazioni. L'ingresso bRetain a TRUE fa in modo che il broker
// mantenga questa pubblicazione a disposizione per i client che si potrebbero 
// collegare in un secondo momento. Questa cosa ha senso visto che i dati 
// pubblicati al cambiamento potrebbero non cambiare per un tempo lungo e si 
// lascerebbe il client senza indicazioni per molto.

FOR udi := 0 TO nOnChangePublishSize - 1 DO
	bIsEqual :=  F_IOT_IsValueEqual(aOnChangePublish[udi].stData.eType, 
									aOnChangePublish[udi].stData.uValue, 
									aOnChangePublish[udi].uOldValue);
	IF bForceOnChangePublish OR NOT bIsEqual THEN
														
		F_IOT_GetPayload(aOnChangePublish[udi].stData, ADR(sPayload), SIZEOF(sPayload));
		fbMqttClient.Publish(
					sTopic:= aOnChangePublish[udi].stData.sSubtopic, 
					pPayload:= ADR(sPayload), 
					nPayloadSize:= LEN2(ADR(sPayload)), 
					eQoS:= TcIotMqttQos.AtMostOnceDelivery, 
					bRetain:= TRUE,								 // !
					bQueue:= FALSE
		);
		aOnChangePublish[udi].uOldValue := aOnChangePublish[udi].stData.uValue;
	END_IF	
END_FOR

bForceOnChangePublish := FALSE;
END_ACTION

ACTION ACT_PublishPeriodic:
(* -----------------------------------------------------------------------------
| This sample has been supplied by Beckhoff As-Is and is intended only as an   |
| example implementation. Functionality is not guaranteed.                     |
----------------------------------------------------------------------------- *)

// Questa Action si occupa della pubblicazione dei dati periodici. Si cicla 
// tra gli elementi dell'array distinguendo tra i dati con pubblicazione veloce
// e quelli a pubblicazione lenta e verificando la presenza del trigger
// corrispondente. Se le condizioni sono soddisfate si calcola il payload con 
// F_IOT_GetPayload che converte il valore del dato in una stringa e  lo si 
// pubblica sul topic con il metodo Public di fbMqttClient.
// L'ingresso eQos indica la qualità richiesta per questa pubblicazione: in
// questo caso si desidera che la pubblicazione avvenga una e una sola volta, 
// senza duplicazioni. L'ingresso bRetain a FALSE fa in modo che il broker non
// mantenga questa pubblicazione a disposizione per i client che si potrebbero 
// collegare in un secondo momento. 

FOR udi := 0 TO nPeriodicPublishSize - 1 DO
	IF fbRtFast.Q AND aPeriodicPublish[udi].eUpdateSpeed = E_IOT_UpdateSpeed.Fast THEN	
		F_IOT_GetPayload(aPeriodicPublish[udi].stData, ADR(sPayload), SIZEOF(sPayload));
		fbMqttClient.Publish(
				sTopic:= aPeriodicPublish[udi].stData.sSubtopic, 
				pPayload:= ADR(sPayload), 
				nPayloadSize:= LEN2(ADR(sPayload)), 
				eQoS:= TcIotMqttQos.AtMostOnceDelivery, 
				bRetain:= FALSE,
				bQueue:= FALSE
		);
	END_IF;	
	
	IF fbRtSlow.Q AND aPeriodicPublish[udi].eUpdateSpeed = E_IOT_UpdateSpeed.Slow THEN	
		F_IOT_GetPayload(aPeriodicPublish[udi].stData, ADR(sPayload), SIZEOF(sPayload));
		fbMqttClient.Publish(
				sTopic:= aPeriodicPublish[udi].stData.sSubtopic, 
				pPayload:= ADR(sPayload), 
				nPayloadSize:= LEN2(ADR(sPayload)), 
				eQoS:= TcIotMqttQos.AtMostOnceDelivery, 
				bRetain:= FALSE,
				bQueue:= FALSE
		);
	END_IF;
END_FOR
END_ACTION

END_FUNCTION_BLOCK

// ---- IOT/Functions/F_IOT_IsValueEqual.TcPOU
(* -----------------------------------------------------------------------------
| This sample has been supplied by Beckhoff As-Is and is intended only as an   |
| example implementation. Functionality is not guaranteed.                     |
----------------------------------------------------------------------------- *)

// Questa funzione confronta il valore attuale del dato con il suo valore 
// precedente.  Anche qui si vede l'utilità dell'unione: se non si fosse 
// utilizzata l'unione sarebbero state necessarie tre  funzioni molto simili 
// che differivano solamente per il tipo di dato in ingresso.

FUNCTION F_IOT_IsValueEqual : BOOL
VAR_INPUT
	eType : E_IOT_DataType;
	uVal1 : U_IOT_DataValue;
	uVal2 : U_IOT_DataValue;	
END_VAR
VAR
END_VAR


IF eType = E_IOT_DataType.Boolean THEN
	F_IOT_IsValueEqual := uVal1.b = uVal2.b;
ELSIF eType = E_IOT_DataType.F64 THEN
	F_IOT_IsValueEqual := uVal1.f = uVal2.f;
ELSIF eType = E_IOT_DataType.I32 THEN
	F_IOT_IsValueEqual := uVal1.n = uVal2.n;
ELSIF eType = E_IOT_DataType.S50 THEN
	F_IOT_IsValueEqual := uVal1.sv = uVal2.sv;	
ELSE
	F_IOT_IsValueEqual := FALSE;	
END_IF

END_FUNCTION

// ---- IOT/Functions/F_IOT_GetPayload.TcPOU
(* -----------------------------------------------------------------------------
| This sample has been supplied by Beckhoff As-Is and is intended only as an   |
| example implementation. Functionality is not guaranteed.                     |
----------------------------------------------------------------------------- *)

// Questa funzione calcola il Payload del dato. Il Payload altro non è che la
// rappresentazione del valore come stringa. Qui si vede l'utilità dell'unione
// se non si fosse utilizziata l'unione sarebbero state necessarie tre 
// funzioni molto simili che differivano solamente per il tipo di dato in 
// ingresso.


FUNCTION F_IOT_GetPayload : BOOL
VAR_INPUT
	stDataValue : ST_IOT_Data;
	pPayload : POINTER TO STRING;
	nSize : UDINT;
END_VAR
VAR
	bRes : BOOL;
	sAppo1 : STRING(255);	
END_VAR

(* -----------------------------------------------------------------------------
| This sample has been supplied by Beckhoff As-Is and is intended only as an   |
| example implementation. Functionality is not guaranteed.                     |
----------------------------------------------------------------------------- *)

IF stDataValue.eType = E_IOT_DataType.Boolean THEN 
	sAppo1 := TO_STRING(stDataValue.uValue.b);
ELSIF stDataValue.eType = E_IOT_DataType.F64 THEN
	sAppo1 := TO_STRING(stDataValue.uValue.f);
ELSIF stDataValue.eType = E_IOT_DataType.S50 THEN
	sAppo1 := stDataValue.uValue.sv;
ELSE
	sAppo1 := TO_STRING(stDataValue.uValue.n);
END_IF
	
F_IOT_GetPayload := STRNCPY(pPayload, ADR(sAppo1), nSize);

END_FUNCTION

// ---- POUs/MAIN.TcPOU
PROGRAM MAIN


VAR
	stRawIn		:	ST_CSL_RawIn;
	stRawOut	:	ST_CSL_RawOut;
	stIn		:	ST_CSL_In;
	stOut		: 	ST_CSL_Out;
	stHMIIn		:	ST_HMI_In;
	stHMIOut	:	ST_HMI_Out;
	stParams	:	ST_CSL_Params;
	stHMIParams	:	ST_HMI_Params; 
	
	fbUpdateInputs	: FB_UpdateInputs;
	fbUpdateOutputs : FB_UpdateOutputs;
	fbUpdateParams	: FB_UpdatesParams;
	
	fbCSL		:	FB_CSL_MAIN;
	
	estep 	: E_Step;
	eErrstep : E_Step;
	
	slot	: INT;
	nerrid	: DINT; 
	bfbend : BOOL;
	
	eSubStepSensor: E_Step;
	eSubStepPistons: E_Step;
	eErrSubStep: E_Step;
	nErrSubId: DINT;
	nTotalRevs: REAL;
END_VAR


fbUpdateParams(stHMIparams := stHMIParams, stParams => stParams);

fbUpdateInputs(stRawIn:= stRawIn, stHMIIn:= stHMIIn, stIn:= stIn);

fbCSL(
	bEnable:= TRUE, 
	stIn:= stIn, 
	stParams:= stParams, 
	stOut:= stOut, 
	eStep=> eStep, 
	eSubStepSensor=> eSubStepSensor,
	eSubStepPistons=> eSubStepPistons, 
	eErrStep=> eErrStep, 
	eErrSubStep=> eErrSubStep, 
	nErrid=> nErrId, 
	nErrSubid=> nErrSubId, 
	bFbEnd=> bFbEnd,
	nTotalRevs => nTotalRevs
);

GVL_PLC.strEStep := TO_STRING(eStep);
GVL_PLC.strEsubStepSensor	:= TO_STRING(eSubStepSensor);
GVL_PLC.strEsubStepPiston	:= TO_STRING(eSubStepPistons);

GVL_PLC.estep := eStep;
GVL_PLC.eSubStepSensor := eSubStepSensor;
GVL_PLC.eSubStepPistons := eSubStepPistons;
GVL_PLC.nColorSensor := stIn.nColorSensor;
GVL_PLC.nTotalRevs	:= fbCSL.nTotalRevs;
GVL_PLC.nCycles	:= fbCSL.nCycles;

fbUpdateOutputs(stOut:= stOut, stRawOut:= stRawOut, stHMIOut => stHMIOut);

END_PROGRAM

// ---- CSL/FB/IO/FB_UpdateInputs.TcPOU
FUNCTION_BLOCK FB_UpdateInputs
VAR_INPUT
	stRawIn		:	ST_CSL_RawIn;	
	stHMIIn		:	ST_HMI_In;
END_VAR
VAR_IN_OUT
	stIn		:	ST_CSL_In;
END_VAR
VAR_OUTPUT
END_VAR
VAR
	
	Filter	:	FB_Filter;
END_VAR

stIn.bMotorImpulse 			:= stRawIn.bMotorImpulse 		;
stIn.bPieceSensorInput 		:= stRawIn.bPieceSensorInput 	;
stIn.bPieceSensorOutput 	:= stRawIn.bPieceSensorOutput 	;	
stIn.bSlot1 				:= stRawIn.bSlot1 				;	
stIn.bSlot2 				:= stRawIn.bSlot2 				;	
stIn.bSlot3	            	:= stRawIn.bSlot3				; 
stIn.bStart 				:= stRawIn.bStart OR stHMIIn.bStart;    	
stIn.bStop					:= stRawIn.bStop AND NOT stHMIIn.bStop;	
stIn.bAck 					:= stRawIn.bAck OR stHMIIn.bAck;
stIn.bEmerg 				:= stRawIn.bEmerg AND stRawIn.bMainEmerg;

Filter(VIn := FC_Conversion(stRawIn.nColorSensor, -10.0, 10.0), VOut := stIn.nColorSensor);

END_FUNCTION_BLOCK

// ---- CSL/FC/FC_Conversion.TcPOU
FUNCTION FC_Conversion : REAL
VAR_INPUT
	I4 		: 	INT;
	Vmin 	: 	REAL;
	Vmax 	:	REAL;
END_VAR
	
VAR
	Rin	: REAL;
END_VAR

VAR CONSTANT
	Livelli	:	REAL	:= 	32767.0;
END_VAR

Rin	:= INT_TO_REAL(I4);
FC_Conversion	:=	Rin/Livelli*(Vmax-Vmin)/2.0;

END_FUNCTION

// ---- CSL/FB/IO/FB_UpdateOutputs.TcPOU
FUNCTION_BLOCK FB_UpdateOutputs
VAR_INPUT
	stOut		: 	ST_CSL_Out;
	
END_VAR
VAR_IN_OUT
	stRawOut	:	ST_CSL_RawOut;
END_VAR
VAR_OUTPUT
	stHMIOut	:	ST_HMI_Out;
END_VAR
VAR
END_VAR

stRawOut.bCompressor := stOut.bCompressor;
stRawOut.bLAck := stOut.bLAck;
stRawOut.bLStart := stOut.bLStart;
stRawOut.bLStop := stOut.bLStop;
stRawOut.bMotor := stOut.bMotor;
stRawOut.bValveSlot1 := stOut.bValveSlot1;
stRawOut.bValveSlot2 := stOut.bValveSlot2;
stRawOut.bValveSlot3 := stOut.bValveSlot3;

(*Comando uscite HMI*)
stHMIOut.bGreen	:= stRawOut.bLStart;
stHMIOut.bRed	:= stRawOut.bLStop;
stHMIOut.bOrange	:= stRawOut.bLAck;

END_FUNCTION_BLOCK

// ---- CSL/FB/IO/FB_UpdatesParams.TcPOU
FUNCTION_BLOCK FB_UpdatesParams
VAR_INPUT
	stHMIparams	:	ST_HMI_Params;
END_VAR
VAR_OUTPUT
	stParams	:	ST_CSL_Params;
END_VAR
VAR
END_VAR

stParams := FC_thresholdsCalculation(stHMIParams := stHMIParams);

stParams.Threshold := stHMIParams.Threshold;

stParams.BlueVoltage	:=	stHMIparams.BlueVoltage;
stParams.RedVoltage		:=	stHMIparams.RedVoltage;
stParams.WhiteVoltage	:=	stHMIparams.WhiteVoltage;

stParams.BlueSlot 	:= stHMIparams.BlueSlot;
stParams.RedSlot  	:= stHMIparams.RedSlot;
stParams.WhiteSlot	:= stHMIparams.WhiteSlot;

END_FUNCTION_BLOCK

// ---- CSL/FC/FC_thresholdsCalculation.TcPOU
FUNCTION FC_thresholdsCalculation : ST_CSL_Params
VAR_INPUT
	stHMIParams : ST_HMI_Params;
END_VAR
VAR
END_VAR

FC_thresholdsCalculation.WhiteVoltageMax	:=	stHMIParams.WhiteVoltage + stHMIParams.Threshold;
FC_thresholdsCalculation.WhiteVoltageMin	:=	stHMIParams.WhiteVoltage - stHMIParams.Threshold;

FC_thresholdsCalculation.RedVoltageMax		:=	stHMIParams.RedVoltage + stHMIParams.Threshold;
FC_thresholdsCalculation.RedVoltageMin		:=	stHMIParams.RedVoltage - stHMIParams.Threshold;

FC_thresholdsCalculation.BlueVoltageMax		:=	stHMIParams.BlueVoltage + stHMIParams.Threshold;
FC_thresholdsCalculation.BlueVoltageMin		:=	stHMIParams.BlueVoltage - stHMIParams.Threshold;

END_FUNCTION

// ---- CSL/FB/Main/FB_CSL_MAIN.TcPOU
FUNCTION_BLOCK FB_CSL_MAIN
VAR_INPUT
	bEnable		:	BOOL;
END_VAR
VAR_IN_OUT
	stIn		:	ST_CSL_In;
	stParams	: 	ST_CSL_Params;
	stOut		:	ST_CSL_Out;
END_VAR
VAR_OUTPUT
	eStep	: E_Step;	//current step of the state machine
	eSubStepSensor: E_Step;
	eSubStepPistons: E_Step;
	eErrStep : E_Step;  //step where an error was raised
	eErrSubStep: E_Step;
	nErrid	: DINT;		//error identification code
	tStepTime : TIME;
	nErrSubid	: DINT;
	
	bFbEnd	: BOOL;
	
	nTotalRevs : REAL;
	
	nCycles : INT;
END_VAR
VAR
	bInitialized	: BOOL;		//FB initialization
	eNewStep : E_Step;			//request for a new step
	bEntryact	: 	BOOL;		//step entry action performed
	fbTonStep :  TON;			// elapsed time on each state machine step
	
	fbSensor	: 	FB_MSF_Sensor;
	fbPiston	:	FB_MSF_Pistons;
	
	fbOscillator:	FB_Oscillator;
	
	fbRestore	:	FB_Restore;
	
	bFbSensorEnd: BOOL;
	bFbPistonEnd: BOOL;
	
	
	nSlot : INT;
	
	Timer_bPause : TON();
	bPause: BOOL	:= FALSE;
	
	bConveyorFree : BOOL;
	iMotorPrev: INT;
	eEmergStep: E_Step;
	
	bFbSensorReset: BOOL;
	bFbPistonsReset: BOOL;
	
	fbRtMotorImpulse: R_TRIG;
	iMotorTotal : INT;
	
END_VAR

(*Initialization of the FB_Sensor*)
IF NOT bInitialized THEN
	eNewStep := E_Step.NoStep;
	eStep := E_Step.MainStop;
	bEntryAct := FALSE;
	bFbEnd := FALSE;
	bInitialized := TRUE;
	bFbSensorReset := TRUE;
	bFbPistonsReset := TRUE;
ELSE
	
	(*Preamble*)
	
	(*Forcing the Not Enabled State*)
	IF NOT bEnable THEN
		eNewStep := E_Step.NeOrError;
	END_IF	
	
	(*Forcing ther emergency state*)
	IF NOT stIn.bEmerg THEN
		IF eStep <> E_Step.MainEmergency THEN
			eEmergStep := eStep;
		END_IF
		eNewStep := E_Step.MainEmergency;
	END_IF
	
	
	(*State change management*)
	IF eNewStep <> E_Step.NoStep THEN
		eStep := eNewStep;
		eNewStep := E_Step.NoStep;
		bEntryact := FALSE;
	END_IF
	
	//bPause management
	(*
	Timer_bPause(IN := NOT stIn.bStop, PT := stParams.stopLongPressTime);
	IF Timer_bPause.Q AND (eStep = E_Step.MainPiston OR eStep = E_Step.MainSensor) THEN
		IF eStep = E_Step.MainSensor AND eSubStepSensor = E_Step.Measuring THEN
			bPause := TRUE;
		ELSE
			eNewStep := E_Step.MainPause;
		END_IF
	END_IF
	*)
	IF NOT stIn.bStop THEN
		bPause := TRUE;
		IF eSubStepSensor = E_Step.Start THEN
			eNewStep := E_Step.MainStop;
		END_IF
	END_IF
	
	fbOscillator(enable := TRUE, t_high := T#500MS, t_low := T#500MS);
	
	//calcolo giri del motori complessivo
	fbRtMotorImpulse(CLK:=	stIn.bMotorImpulse );
	IF fbRtMotorImpulse.Q THEN
		iMotorTotal := iMotorTotal + 1;
		nTotalRevs := TO_REAL(iMotorTotal) / 4;
	END_IF
	
	(* msf subordinate *)
	fbSensor(
		bInitializedExt := TRUE,
		stIn:= stIn, 
		bEnable:= bEnable,
		bRun:= (eStep = E_Step.MainSensor), 
		eStep=> eSubStepSensor, 
		eErrStep=> eErrSubStep, 
		nErrId=> nErrSubId,
		bFbEnd=> bFbSensorEnd, 
		stOut:= stOut, 
		nSlot=> nSlot, 
		stParams:= stParams
	);
	
	fbPiston(
		bInitializedExt := TRUE,
		bEnable:= bEnable, 
		slot:= nSlot, 
		stIn:= stIn, 
		bRun := (eStep = E_Step.MainPiston),
		stParams:= stParams, 
		stOut:= stOut, 
		eStep=> eSubStepPistons, 
		eErrStep=> eErrSubStep, 
		nErrid=> nErrSubId, 
		iMotorPrev => iMotorPrev,
		bFbEnd=> bFbPistonEnd,
		nCycles=>nCycles
	);

	(*Case*)
	CASE eStep OF
		
		(*MainStop Step - S0*)
		E_Step.MainStop :
			(*Body*)
			bPause := FALSE;
			
			stOut.bLStart	:= fbOscillator.q;
			stOut.bLStop := TRUE;
			stOut.bLAck := FALSE;
			stOut.bMotor:=FALSE;
		
			(*Transition - to MainSensor*)
			IF stIn.bStart AND bEnable THEN
				eNewStep := E_Step.MainSensor;
			END_IF
			
			(*Exit Act*)
			IF eNewStep <> E_Step.NoStep THEN
				IF eNewStep = E_Step.NeOrError THEN
					eErrStep := eStep;
					//nErrId	:= 16#9999_9999;
				END_IF
			END_IF
			
		(*MainSensor Step - S1*)
		E_Step.MainSensor :
			(*Body*)
			stOut.bLStart	:= TRUE;
			stOut.bMotor := fbSensor.bMotor OR fbPiston.bMotor;
			IF bPause THEN
				stOut.bLStop := fbOscillator.q;
			ELSE
				stOut.bLStop := FALSE;
			END_IF
			stOut.bLAck := FALSE;
		(*
			fbSensor(
				bInitializedExt := NOT bFbSensorReset,
				stIn:= stIn, 
				bEnable:= bEnable, 
				eStep=> eSubStep, 
				eErrStep=> eErrSubStep, 
				nErrId=> nErrSubId,
				bFbEnd=> bFbSensorEnd, 
				stOut:= stOut, 
				nSlot=> nSlot, 
				stParams:= stParams
			);
			*)
			
			//bFbSensorReset := FALSE;
			
			(*Transition - to Processing*)
			IF bFbSensorEnd AND bEnable THEN
				eNewStep := E_Step.MainPiston;
			END_IF
			
			(*Exit Act*)
			IF eNewStep <> E_Step.NoStep THEN
				IF eNewStep = E_Step.NeOrError THEN
					eErrStep := eStep;
					//nErrId	:= 16#9999_9999;
				END_IF
				
				bFbSensorReset := FALSE;
			END_IF
		
		(*MainPiston Step - S2*)
		E_Step.MainPiston :
			(*Body*)
			stOut.bLStart	:= TRUE;
			stOut.bMotor := fbSensor.bMotor OR fbPiston.bMotor;
			IF bPause THEN
				stOut.bLStop := fbOscillator.q;
			ELSE
				stOut.bLStop := FALSE;
			END_IF
			stOut.bLAck := FALSE;
		
			
(*
			fbPiston(
				bInitializedExt := NOT bFbPistonsReset,
				bEnable:= bEnable, 
				slot:= nSlot, 
				stIn:= stIn, 
				stParams:= stParams, 
				stOut:= stOut, 
				eStep=> eSubStep, 
				eErrStep=> eErrSubStep, 
				nErrid=> nErrSubId, 
				iMotorPrev => iMotorPrev,
				bFbEnd=> bFbPistonEnd
			);
			*)
			
			//bFbPistonsReset := FALSE;
			
			(*Transition - to MainSensor*)
			(*Transition - to MainPause*)
			IF bFbPistonEnd AND bEnable THEN
				IF bPause THEN
					eNewStep := E_Step.MainStop; //to MainStop
				ELSE
					eNewStep := E_Step.MainSensor; //to MainSensor
				END_IF	
			END_IF
			
			
			(*Exit Act*)
			IF eNewStep <> E_Step.NoStep THEN
				IF eNewStep = E_Step.NeOrError THEN
					eErrStep := eStep;
					//nErrId	:= 16#9999_9999;
				END_IF
			END_IF	
			
		(*MainPause Step - S3*)
		E_Step.MainPause :
			(*Body*)
			stOut.bLStart	:= FALSE;
			stOut.bLStop := TRUE;
			stOut.bLAck := FALSE;
			stOut.bMotor:=FALSE;
			
			(*Transition - to MainSensor*)
			IF stIn.bStart AND bEnable THEN
				eNewStep := E_Step.MainSensor;
				bPause := FALSE;
			END_IF
			
			(*Exit Act*)
			IF eNewStep <> E_Step.NoStep THEN
				IF eNewStep = E_Step.NeOrError THEN
					eErrStep := eStep;
					//nErrId	:= 16#9999_9999;
				END_IF
			END_IF	
		
		(*MainEmergency Step - S4*)
		E_Step.MainEmergency :	
			(*Body*)
			stOut.bLStart	:= FALSE;
			stOut.bLStop := FALSE;
			stOut.bLAck := fbOscillator.q;
			stOut.bMotor:=FALSE;
			
			//da vedere il pilotaggio delle uscite: motore, compressore e valvole
			stOut.bMotor := FALSE;
			stOut.bCompressor := FALSE;
		
			(*Transition - to Measuring*)
			IF stIn.bAck AND bEnable THEN
				eNewStep := E_Step.MainAcknowledge;
			END_IF
			
			(*Exit Act*)
			IF eNewStep <> E_Step.NoStep THEN
				IF eNewStep = E_Step.NeOrError THEN
					eErrStep := eStep;
					//nErrId	:= 16#9999_9999;
				END_IF
			END_IF
			
		(*MainAcknowledge Step - S5*)	
		E_Step.MainAcknowledge :		
			(*Body*)
			stOut.bLStart	:= FALSE;
			stOut.bLStop := FALSE;
			stOut.bLAck := TRUE;
			
			//fb per liberare il nastro
			fbRestore(
				bEnable:= TRUE, 
				iMotorPrev:= iMotorPrev, 
				eStep:= eEmergStep, 
				eSubStepSensor:= eSubStepSensor,
				eSubStepPistons:= eSubStepPistons,
				stIn:= stIn, 
				stParams:= stParams, 
				stOut:= stOut, 
				bFbEnd=> bConveyorFree
			);
		
			(*Transition - to Measuring*)
			IF bConveyorFree AND bEnable THEN
				bInitialized := FALSE;
				iMotorPrev := 0;
			END_IF
			
			(*Exit Act*)
			IF eNewStep <> E_Step.NoStep THEN
				IF eNewStep = E_Step.NeOrError THEN
					eErrStep := eStep;
					//nErrId	:= 16#9999_9999;
				END_IF
			END_IF
		
		(*NeOrError step*)	
		E_Step.NeOrError :
			(*Body*)
			stOut.bLStart	:= fbOscillator.q;
			stOut.bLStop := fbOscillator.q;
			stOut.bLAck := fbOscillator.q;
			
			stOut.bMotor := FALSE;
		
			(*Transition - to Measuring*)
			
			
			(*Exit Act*)
			IF eNewStep <> E_Step.NoStep THEN
				IF eNewStep = E_Step.NeOrError THEN
					eErrStep := eStep;
					//nErrId	:= 16#9999_9999;
				END_IF
			END_IF
			
	END_CASE
	
		(* elapsed time into the current step *)
	fbTonStep(IN := (eNewstep = E_Step.NoStep), PT := T#500H);
	tStepTime := fbTonStep.ET;
END_IF

END_FUNCTION_BLOCK

// ---- CSL/FB/Sensor/FB_MSF_Sensor.TcPOU
FUNCTION_BLOCK FB_MSF_Sensor
VAR_INPUT

	bEnable				:	BOOL;
	bRun				: BOOL;
	bInitializedExt	:	BOOL;
	
END_VAR

VAR_OUTPUT
	eStep				:	E_Step;
	eErrStep			:	E_Step;
	nErrId				:	DINT;
	
	bFbEnd				:	BOOL;

	nSlot				:	INT;

	bMotor				:	BOOL;	
END_VAR

VAR_IN_OUT
	stIn		:	ST_CSL_In;
	stParams	: 	ST_CSL_Params;
	stOut		: 	ST_CSL_Out;	
	
END_VAR

VAR
	bInitialized		:	BOOL;
	eNewStep			:	E_Step;
	bEntryAct			:	BOOL;
	fbTonStart			:	TON;
	
	fbMeasure			:	FB_Measuring;
	fbSlot				:	FB_Processing;
	
	
	rPieceValue			:	REAL;
	bEndMeasure			:	BOOL;
	
END_VAR

(*Initialization of the FB_Sensor*)
IF NOT bInitialized OR NOT bInitializedExt THEN
	eNewStep := E_Step.NoStep;
	eStep := E_Step.Stop;
	bEntryAct := FALSE;
	bFbEnd := FALSE;
	bInitialized := TRUE;
ELSE
	
	(*Preamble*)
	
	(*Forcing the Error State*)
	IF NOT bEnable THEN
		eNewStep := E_Step.NeOrError;
	END_IF	
	
	(*State change management*)
	IF eNewStep <> E_Step.NoStep THEN
		eStep := eNewStep;
		eNewStep := E_Step.NoStep;
		bEntryact := FALSE;
	END_IF
	
	(*Filters*)
	fbTonStart(IN := NOT stIn.bPieceSensorInput, PT := T#2S);
		
	(*Case*)
	CASE eStep OF
		(*Stop Step*)
		E_Step.Stop :
			(*Body*)
			bMotor := FALSE;
		
			(*Transition - to Measuring*)
			IF bRun AND bEnable THEN
				eNewStep := E_Step.Start;
			END_IF
			
			(*Exit Act*)
			IF eNewStep <> E_Step.NoStep THEN
				IF eNewStep = E_Step.NeOrError THEN
					eErrStep := eStep;
					//nErrId	:= 16#9999_9999;
				END_IF
			END_IF		
	
		(*Start Step*)
		E_Step.Start :
			(*Body*)
			bMotor := FALSE;
		
			(*Transition - to Measuring*)
			IF fbTonStart.Q AND bEnable THEN
				eNewStep := E_Step.Measuring;
			END_IF
			
			(*Exit Act*)
			IF eNewStep <> E_Step.NoStep THEN
				IF eNewStep = E_Step.NeOrError THEN
					eErrStep := eStep;
					//nErrId	:= 16#9999_9999;
				END_IF
			END_IF
			
		(*Measuring Step*)
		E_Step.Measuring :
			(*Body*)
			bMotor := TRUE;
		
			fbMeasure(Vin := stIn.nColorSensor, Vout := rPieceValue);
			
			(*Transition - to Processing*)
			IF NOT stIn.bPieceSensorOutput AND bEnable THEN
				fbSlot(SensorInput := rPieceValue, stParams := stParams);
				nSlot := fbSlot.slot;
				eNewStep:=E_Step.Stop;
				bInitialized := FALSE;
				bFbEnd := TRUE;
			END_IF
			
			(*Exit Act*)
			IF eNewStep <> E_Step.NoStep THEN
				IF eNewStep = E_Step.NeOrError THEN
					eErrStep := eStep;
					//nErrId	:= 16#9999_9999;
				END_IF
			END_IF
		
		E_Step.NeOrError :
			(*Body*)
			bMotor := FALSE;
		
			bInitialized := FALSE;
			
			(*Exit Act*)
			IF eNewStep <> E_Step.NoStep THEN
				IF eNewStep = E_Step.NeOrError THEN
					eErrStep := eStep;
					//nErrId	:= 16#9999_9999;
				END_IF
			END_IF
			
	END_CASE
END_IF

END_FUNCTION_BLOCK

// ---- CSL/FB/Sensor/FB_Measuring.TcPOU
FUNCTION_BLOCK FB_Measuring
VAR_INPUT
	VIn		:	REAL;
END_VAR
VAR_OUTPUT
	EndMeasure	:	BOOL;
	
END_VAR
VAR_IN_OUT
	VOut		:	REAL;
END_VAR
VAR
	VPrev	:	REAL	:=	10.0;
	fbTonEndMeasure	:	TON;
	En : BOOL;
END_VAR

IF VIn < VPrev OR VIn > 7.3 THEN
    VPrev := VIn;
    En := VIn < VPrev; (* En sarà TRUE solo se VIn < VPrev *)
END_IF

IF En THEN
    Vout := VPrev;
END_IF

END_FUNCTION_BLOCK

// ---- CSL/FB/Sensor/FB_Processing.TcPOU
FUNCTION_BLOCK FB_Processing
VAR_INPUT
	SensorInput	:	REAL;
END_VAR
VAR_OUTPUT
	slot		:	INT;
	
END_VAR
VAR_IN_OUT
	stParams	:	ST_CSL_Params;	
END_VAR
VAR
END_VAR

IF SensorInput < stParams.BlueVoltageMax AND SensorInput > stParams.BlueVoltageMin THEN
	slot	:=	stParams.BlueSlot;
ELSIF SensorInput < stParams.RedVoltageMax AND SensorInput > stParams.RedVoltageMin THEN
	slot	:=	stParams.RedSlot;
ELSIF SensorInput < stParams.WhiteVoltageMax AND SensorInput > stParams.WhiteVoltageMin THEN
	slot	:=	stParams.WhiteSlot;
ELSE
	slot	:=	0;
END_IF

END_FUNCTION_BLOCK

// ---- CSL/FB/Piston/FB_MSF_Pistons.TcPOU
FUNCTION_BLOCK FB_MSF_Pistons
VAR_INPUT
	bEnable	: BOOL;  // machine enable
	bInitializedExt	:	BOOL;
	bRun: BOOL;
	slot	: INT;   // destination slot
END_VAR

VAR_IN_OUT
	stIn		:	ST_CSL_In;
	stParams	: 	ST_CSL_Params;
	stOut		: 	ST_CSL_Out;	
END_VAR

VAR_OUTPUT
	eStep	: E_Step;	//current step of the state machine
	eErrStep : E_Step;  //step where an error was raised
	nErrid	: DINT;		//error identification code
	
	iMotorPrev	: INT;         // steps done while travelling on conveyor
	
	bFbEnd	: BOOL;
	
	bMotor	: BOOL;
	
	nCycles : INT;
END_VAR

VAR
	bSensor: BOOL;
	bValve : BOOL;
	nStepSlot : INT;
	Error: DINT;
	iMotor	: INT := 0;         // steps done while travelling on conveyor
    
	bInitialized	: 	BOOL;		//FB initialization
	
	eNewStep : E_Step;			//request for a new step
	bEntryact	: 	BOOL;		//step entry action performed
	
	Timer_Pistons : TON();	
	Timer_WaitingTransition : TON();
	
	Timer_Positioned : TON();
	
	fbRtMotorImpulse : R_TRIG;  // edge detection on conveyor encoder
	
	bSlotFree: BOOL;

END_VAR

(* initialization *)
IF NOT bInitialized OR NOT bInitializedExt THEN    
	eNewstep 		:= 	E_Step.NoStep;    
	eStep 			:= 	E_Step.Stop;    
	bEntryact 		:= 	FALSE;    
	bInitialized 	:= 	TRUE; 
	bSlotFree		:=	FALSE;
	bFbEnd			:=	FALSE;

ELSE   

	(* forcing the error state *)	
	(* disabled or faulty *)
	IF  NOT bEnable THEN
		eNewstep 	:=	E_Step.NeOrError;
	END_IF;

	(* state change management *)
	IF eNewstep <> E_Step.NoStep THEN    
		eStep 		:= 	eNewstep;    
		eNewstep 	:= 	E_Step.NoStep;   
 		bEntryact 	:= 	FALSE;
	END_IF;

	
	(* input signal conditioning *)
	(*filters*)
	Timer_Pistons (IN:= (iMotor = nStepSlot AND eStep = E_Step.waiting), PT := stParams.pistonReentryDelay);
	
	Timer_WaitingTransition (IN := (Timer_Pistons.Q AND eStep = E_Step.waiting), PT := stParams.slotRemoveTime);
	
	Timer_Positioned(IN := (eStep = E_Step.piston), PT := T#100MS);
	
	(*edges*)
	fbRtMotorImpulse(CLK:=	stIn.bMotorImpulse );
	
	// association of the motors and the sensors to the steps
	CASE slot OF
		0:
			nStepSlot	:=	stParams.StepNoSlot;	
		1:
			stOut.bValveSlot1 := bValve;
			bSensor 	:= 	stIn.bSlot1;
			nStepSlot 	:= 	stParams.StepSlot1;
		2:
			stOut.bValveSlot2 := bValve;
			bSensor 	:= 	stIn.bSlot2;
			nStepSlot 	:= 	stParams.StepSlot2;
		3:
			stOut.bValveSlot3 := bValve;
			bSensor 	:= 	stIn.bSlot3;
			nStepSlot 	:= 	stParams.StepSlot3;
			
	END_CASE

	// storing of the pieces
	CASE eStep OF
		(*Stop Step*)
		E_Step.Stop :
			(*Body*)
			bMotor := FALSE;
			iMotor := 0;
			
			bFbEnd := FALSE;
			
			(*Transition - to Measuring*)
			IF bRun AND bEnable THEN
				eNewStep := E_Step.conveyor;
			END_IF
			
			(*Exit Act*)
			IF eNewStep <> E_Step.NoStep THEN
				IF eNewStep = E_Step.NeOrError THEN
					eErrStep := eStep;
					//nErrId	:= 16#9999_9999;
				END_IF
			END_IF		
	
		// a new piece was placed on the conveyor belt
		E_Step.conveyor :
	
			(* body *)	
			IF slot <> 0 THEN
				bMotor		:=	 bSensor;
				stOut.bCompressor 	:=	 bSensor;
			ELSE
				bMotor	:=	TRUE;
				stOut.bCompressor := FALSE;
			END_IF
			
			IF slot <> 0 THEN
				bValve :=	 FALSE;	
			END_IF
			
			(* Update steps Counter *)
			IF fbRtMotorImpulse.Q	THEN
				iMotor := iMotor + 1;
				iMotorPrev := iMotor;
			END_IF
		
			(* transition *)	
			IF NOT bEnable THEN          
		 		eNewstep := E_Step.NeOrError;        
			ELSE 
				IF  iMotor = nStepSlot AND nStepSlot <> stParams.StepNoSlot THEN 
					eNewstep := E_Step.piston;
				ELSIF iMotor = nStepSlot AND nStepSlot = stParams.StepNoSlot THEN
					eNewstep := E_Step.waiting;
        		END_IF;
			END_IF
	
		// activation of the selected piston until the piece falls in its slot
		E_Step.piston :

			(* body *)
			bMotor		:= 	FALSE;
			stOut.bCompressor 	:= 	TRUE;
			IF slot <> 0 AND Timer_Positioned.Q THEN
				bValve :=	TRUE;
			END_IF
	
			(* transition *)
			IF NOT bEnable THEN          
		 		eNewstep := E_Step.NeOrError;        
			ELSE 
				IF NOT bsensor THEN 
					eNewstep := E_Step.waiting;
       	 		END_IF;
			END_IF

		// wait the piston re-entry
		E_Step.waiting :
	
			(* body *)
			bMotor		:=	FALSE;
			stOut.bCompressor 	:= 	FALSE;
			IF slot <> 0 THEN
				bValve :=	FALSE;	
			END_IF
		
			(* transition - to exit *)
			IF NOT bEnable THEN          
		 		eNewstep := E_Step.NeOrError;        
			ELSE 
				IF Timer_WaitingTransition.Q THEN 
					nCycles := nCycles +1;
					eNewstep := E_Step.Stop;
					bFbEnd	:= TRUE; 					           
       	 		END_IF;
			END_IF	
			
		E_Step.NeOrError :
			(*Body*)
			bMotor := FALSE;
		
			bInitialized := FALSE;
			
			
			(*Exit Act*)
			IF eNewStep <> E_Step.NoStep THEN
				IF eNewStep = E_Step.NeOrError THEN
					eErrStep := eStep;
					//nErrId	:= 16#9999_9999;
				END_IF
			END_IF		
			
		ELSE
	
		// Error case
		eNewstep 	:= 	E_Step.NeOrError;
		eErrStep 	:=	E_Step.Unknown;
		nErrId 		:= 	-9; 	
		
		
	END_CASE


END_IF

END_FUNCTION_BLOCK

// ---- CSL/FB/Main/FB_Oscillator.TcPOU
FUNCTION_BLOCK FB_Oscillator
VAR_INPUT
	enable	: BOOL;
	t_high	: TIME;
	t_low	: TIME;	
END_VAR
VAR_OUTPUT
	q		: BOOL;	
END_VAR
VAR
	t1		: TON();
	t2		: TON();	
END_VAR

t1(in := enable AND NOT t2.Q, pt := t_low);
t2(in := t1.Q, pt := t_high);
// comando dell'uscita dell'oscillatore
q := t1.Q;

END_FUNCTION_BLOCK

// ---- CSL/FB/Main/FB_Restore.TcPOU
FUNCTION_BLOCK FB_Restore
VAR_INPUT
	bEnable : BOOL;
	iMotorPrev 		: 	INT;
	eStep		:	E_Step;
	eSubStepSensor	:	E_Step;
	eSubStepPistons	:	E_Step;
END_VAR
VAR_IN_OUT
	stIn		:	ST_CSL_In;
	stParams	: 	ST_CSL_Params;
	stOut		:	ST_CSL_Out;
END_VAR
VAR_OUTPUT
	bFbEnd		:	BOOL;
END_VAR
VAR
	iMotor		:	INT;

	bPieceOut 	:	BOOL;	

	fbRtMotorImpulse : R_TRIG;
	
	bInitialized: BOOL;
END_VAR


IF NOT bInitialized THEN
	bFbEnd := FALSE;
	bInitialized := TRUE;
	bPieceOut := FALSE;
	iMotor := 0;
ELSE
	IF eSubStepSensor = e_Step.Start THEN
		bInitialized := FALSE;
		bFbEnd := TRUE;
	END_IF
	IF eStep = E_Step.MainSensor AND NOT bPieceOut THEN
		stOut.bMotor := TRUE;
		IF NOT stIn.bPieceSensorOutput AND bEnable THEN
			bPieceOut := TRUE;
		END_IF	
	ELSIF eStep = E_Step.MainPiston  OR bPieceOut THEN
		stOut.bMotor := TRUE;
	
		fbRtMotorImpulse(CLK:=	stIn.bMotorImpulse );
		
		IF fbRtMotorImpulse.Q	THEN
			iMotor := iMotor + 1;
		END_IF
			
		IF iMotor = (stParams.StepNoSlot - iMotorPrev ) THEN
			stOut.bMotor := FALSE;
			bInitialized := FALSE;
			bFbEnd := TRUE;
		END_IF

	ELSE
		bInitialized := FALSE;
		bFbEnd := TRUE;
	END_IF
END_IF

END_FUNCTION_BLOCK
